(* IEC 61131-3 sources: volt/packages/volt-lsp-iec/test-corpus/lenze-mid/Device/Plc Logic/Application/Library Manager/L_OEEA_MachinePerformanceSolution, 3.26.4.18 (Lenze), 18 files *)

(* ---- SCCUTTHROUGPUTAVERAGELREAL.dut ---- *)
TYPE SCCUTTHROUGPUTAVERAGELREAL :
STRUCT
	LRREALINPUTVALUE : LREAL;
	LRINAVGVALUE : LREAL;
	SCUTREALSTR : STRING;
	LRCUTREAL : LREAL;
	IARRAYINDEX : INT;
	ALRVALUEARRAY : ARRAY [0..60] OF LREAL;
	LRAVERAGEVALUE : LREAL;
	LRLASTREALVALUE : LREAL;
	XARRAYFILLEDONCE : BOOL;
END_STRUCT
END_TYPE

(* ---- SCTREND_LIMITS.dut ---- *)
TYPE SCTREND_LIMITS :
STRUCT
	LRUPPERLIMIT : LREAL;
	DIUPPERROUNDLIMIT : DINT;
	DIMIDDLEROUNDLIMIT : DINT;
	DIFACTOR : INT;
	XTARGETUPPER : BOOL;
END_STRUCT
END_TYPE

(* ---- VERSIONCONSTANTS.gvl ---- *)
VAR_GLOBAL
	GC_BYAMOUNTOFGENERALDATA : BYTE := 50;
	GC_BYAMOUNTDOWNTIMEERRORS : BYTE := 10;
	GC_IFILTERSAMPLES : INT := 20;
END_VAR

(* ---- CALACTUALALLTIME.pou ---- *)
FUNCTION CALACTUALALLTIME : TIME
VAR_INPUT
	DTCURRENTTIME : TIME_OF_DAY;
	DTSETWEEKSTARTTIME : TIME_OF_DAY;
	EACTUALWEEKDAY : RTCLK.WEEKDAY;
	ESETWEEKDAY : RTCLK.WEEKDAY;
END_VAR
END_FUNCTION

(* ---- CALAVERARGELREALSUMMERYVALUE.pou ---- *)
FUNCTION CALAVERARGELREALSUMMERYVALUE : LREAL
VAR_INPUT
	LRVALUE : LREAL;
	INOOFAVERAGECOUNT : INT;
END_VAR
VAR_IN_OUT
	SCCUTAVERAGEREAL : scCutThrougputAveragelReal;
END_VAR
END_FUNCTION

(* ---- XYTRENDUPPERLIMIT.pou ---- *)
FUNCTION XYTRENDUPPERLIMIT : scTrend_Limits
VAR_INPUT
	LRTARGETVALUE : LREAL;
	LRACTUALVALUE : LREAL;
END_VAR
END_FUNCTION

(* ---- FBPROLONGTIME.pou ---- *)
FUNCTION_BLOCK FBPROLONGTIME
VAR_INPUT
	TPROLONGTIME : TIME;
	XSTARTPROLONGTIME : BOOL;
END_VAR
VAR_OUTPUT
	XPROLONG : BOOL;
END_VAR
VAR
	TONPROLONGTIMER : TON;
	TRIGPROLONG : R_TRIG;
END_VAR
END_FUNCTION_BLOCK

(* ---- L_OEEA_BASE.pou ---- *)
FUNCTION_BLOCK L_OEEA_BASE
VAR_INPUT
	XENABLE : BOOL;
	XRESET : BOOL;
END_VAR
VAR_IN_OUT
	SCSHIFTVALUES : scCurrentShiftValues;
	SCPDINTERNAL : scInternalVar;
END_VAR
VAR
	XACTIVELICENSE : BOOL := TRUE;
	XFIRSTCYCLE : BOOL := FALSE;
	I : INT;
	SCSHIFTCHANGEPERFORMANCE : scPerformance_base;
	SCSHIFTCHANGESCAP : scAccessPoints;
	SCINTERNSHIFTVALUES : scCurrentShiftValues;
	PUIHOUR : UINT;
	PUIHOUR2 : UINT;
	PUIHOUR3 : UINT;
	PUIHOUR4 : UINT;
	PUIHOUR5 : UINT;
	PUIMINUTE : UINT;
	PUIMINUTE2 : UINT;
	PUIMINUTE3 : UINT;
	PUIMINUTE4 : UINT;
	PUIMINUTE5 : UINT;
	PUISECOND : UINT;
	PUISECOND2 : UINT;
	PUISECOND3 : UINT;
	PUISECOND4 : UINT;
	PUISECOND5 : UINT;
	PUIMILLISECOND : UINT;
	PUIMILLISECOND2 : UINT;
	PUIMILLISECOND3 : UINT;
	PUIMILLISECOND4 : UINT;
	PUIMILLISECOND5 : UINT;
	XERROR : DTU.Error;
	XERROR2 : DTU.Error;
	XERROR3 : DTU.Error;
	LRPROGRESSIVETARGET : LREAL;
	SCPDINTERNALCLEAR : scInternalVar;
	XSHIFTRESET : BOOL;
	XINCONSISTENTDATARESET : BOOL;
	DTDAYCHANGETIME : TIME_OF_DAY;
	DTSTARTRECORDDATETIME : DATE_AND_TIME := DATE_AND_TIME#1970-1-1-0:0;
	FTXACTIVESHIFT : F_TRIG;
	FT_XRESET : R_TRIG;
	RTSHIFT0 : R_TRIG;
	RS_XRESET : RS;
	RTDOWNTIMECOUNT : R_TRIG;
	RTCALLFORSERVICE : R_TRIG;
	FBRRTIMER : TON;
	FBCALLFORSERVICE : TON;
	FBOEEKPISTIMEEVENT : TON;
	FBOEEKPIPROLONGED : TON;
	ILASTPRODUCTIONMODE : INT;
	ILASTDOWNTIMECATEGORY : INT;
	IPREVPRODUCTIONMODE : INT;
	IPREVDOWNTIMECATEGORY : INT;
	UDILASTDOWNTIMEREASON : UDINT;
	UDIPREVDOWNTIMEREASON : UDINT;
	IWEEKDAYDIFF : INT;
	XDEACTIVESHIFTCONTINIOUSUPDATE : BOOL;
	XSHIFTRESETEVENTDELAY : BOOL;
	XSHIFTRESETEVENTDELAYDONE : BOOL;
	FBACTUALPARTCOUNT : TON_Pausable;
	XRESETPRODUCTTYPEDATA : BOOL;
	T100MSTIMER : TON;
	DTCURRENTTIME : TIME_OF_DAY;
	XSTATECHANGEDETECTED : BOOL;
	FTRIGENDWAITINGTIMEPOWERONCYCLE : F_TRIG;
	RLASTTECHNICALCYCLETIME : REAL;
	RPARTTARGET_ACT : REAL;
	RTIMEDELTA : REAL;
	RLASTTARGETOEE : REAL;
	XSTATECHANGEAFTERPOWERCYCLE : BOOL;
	FBSTATECHANGEAFTERPOWERCYCLE : TON;
	XSTATECHANGEWAITINGTIME : BOOL;
	XSTATECHANGEDETECTEDONECYCLE : BOOL;
	SCIN_BATCHPRODUCTEND : scBatchProductEnd;
	SCBATCHPRODUCTEND : scBatchProductEnd;
	XFTXACTIVESHIFTDETECTED : BOOL;
	XHALTTIMETRIGGER : BOOL;
	THALTTIMETRIGGER : TIME;
	TONPROLONGTIMER : ARRAY [1..2] OF TON;
	ISTEPSHIFTCHANGE : INT := 0;
	XEVENTPROLONG : BOOL;
	XWAITPROLONG : BOOL;
	XSTATECHANGEPROLONGED : BOOL;
	FBSTATECHANGE : fbProlongTime;
	FBSTATECHANGEWAIT : fbProlongTime;
	XSEQSTATECHANGEBUSY : BOOL;
	XPRODUCTIONEVENTMODE : BOOL;
	XRESETDEACTIVESHIFTCONTINIOUSUPDATE : BOOL;
	XSETDEACTIVESHIFTCONTINIOUSUPDATE : BOOL;
END_VAR
END_FUNCTION_BLOCK

METHOD ACT_MAIN_BASE : BOOL
VAR_INPUT
	SCTRIGGER : scTrigger_base;
	EOEECALCMODE : enumOEECalculationMode;
	IPRODUCTIONEVENTMODE : INT;
END_VAR
VAR_IN_OUT
	SCMACHINEDATA : scMachineData_base;
	SCSHIFTVALUES : scCurrentShiftValues;
	SCSHIFTPERFORMANCE : scPerformance_base;
	SCPDINTERNAL : scInternalVar;
END_VAR
END_METHOD

METHOD ACT_PARTCOUNTER : BOOL
VAR_IN_OUT
	SCMACHINEDATA : scMachineData_base;
	SCSHIFTVALUES : scCurrentShiftValues;
	SCSHIFTPERFORMANCE : scPerformance_base;
	SCPDINTERNAL : scInternalVar;
END_VAR
END_METHOD

METHOD ACT_SHIFTCHANGEEVENT : BOOL
VAR_IN_OUT
	SCMACHINEDATA : scMachineData_base;
	SCSHIFTVALUES : scCurrentShiftValues;
	SCSHIFTPERFORMANCE : scPerformance_base;
	SCPDINTERNAL : scInternalVar;
END_VAR
END_METHOD

METHOD CAL_PRODUCTIONLOSSES : BOOL
VAR_INPUT
	EOEECALCMODE : enumOEECalculationMode;
END_VAR
VAR_IN_OUT
	SCMACHINEDATA : scMachineData_base;
	SCSHIFTVALUES : scCurrentShiftValues;
	SCPDINTERNAL : scInternalVar;
END_VAR
END_METHOD

METHOD SET_SHIFTDATA : BOOL
VAR_INPUT
	SCTRIGGER : scTrigger_base;
	IPRODUCTIONEVENTMODE : INT;
END_VAR
VAR_IN_OUT
	SCMACHINEDATA : scMachineData_base;
	SCSHIFTVALUES : scCurrentShiftValues;
	SCSHIFTPERFORMANCE : scPerformance_base;
	SCPDINTERNAL : scInternalVar;
END_VAR
END_METHOD

METHOD CAL_PRODUCTIONKPIS : BOOL
VAR_INPUT
	EOEECALCMODE : enumOEECalculationMode;
END_VAR
VAR_IN_OUT
	SCMACHINEDATA : scMachineData_base;
	SCSHIFTPERFORMANCE : scPerformance_base;
	SCPDINTERNAL : scInternalVar;
END_VAR
END_METHOD

METHOD METH_PROLONGBIT : BOOL
VAR_INPUT
	TPROLONGTIME : TIME;
END_VAR
VAR_IN_OUT
	TONPROLONGTIMER : TON;
	XSTARTPROLONGTIME : BOOL;
END_VAR
END_METHOD

(* ---- L_OEEA_CLOUDIF_NA.pou ---- *)
FUNCTION_BLOCK L_OEEA_CLOUDIF_NA
VAR_INPUT
	SDOWNTIMEBITSTR : STRING;
	SCTRIGGER : scTrigger;
	XENABLE : BOOL;
END_VAR
VAR_OUTPUT
	SCCLOUD : scCloud;
END_VAR
VAR_IN_OUT
	SCMACHINEDATA : scMachineData;
	SCPERFORMANCE : scPerformance;
END_VAR
VAR
	FBTRIGGER_SETTINGS : TON;
	FBTRIGGER_RR : TON;
	FBTRIGGER2_SETTINGS : TON;
	FBTRIGGER2_RR : TON;
	FBFIRSTSTARTTRIGGER : TON;
	XFIRSTCYCLE : BOOL;
	XFIRSTTRIGGER : BOOL;
END_VAR
END_FUNCTION_BLOCK

METHOD ACT_MAPVARIABLE
END_METHOD

METHOD ACT_TRIGGERVARIABLE
END_METHOD

(* ---- L_OEEA_DATASIMULATOR.pou ---- *)
FUNCTION_BLOCK L_OEEA_DATASIMULATOR
VAR_INPUT
	XENABLE : BOOL;
	PA_TIMER : RT_Timer;
	XMATERIALPRODUCTION : BOOL;
	RLINESPEED : REAL;
	IPARTCOUNTNOK : INT;
	IINPRODUCTIONMODE : INT;
	INOOFERRORINDEX : INT;
	LRMATERIALCOUNT : LREAL;
END_VAR
VAR_IN_OUT
	SCRT_STATUS_RECORD : RT_Status_Struct;
	SCSHIFTVALUES : scCurrentShiftValues;
	PA_DOWNTIME : RT_Downtime;
END_VAR
VAR
	FBTONALIVE : TON;
	FBR_TRIG_ALIVE : R_TRIG;
	FBTONOK_PARTS : TON;
	FBR_TRIG_OK_PARTS : R_TRIG;
	FBTONNOK_PARTS : TON;
	FBR_TRIG_NOK_PARTS : R_TRIG;
	FBTONERROR : TON;
	FBTONERRORDURATION : TON;
	FBTONPARTCYCLETIME : TON;
	FBTONOPCYCLETIME : TON;
	ERROR_INDEX : INT := 0;
	XERRORDETECTED : BOOL;
	LRAVERAGECYCLETIME : LREAL;
	DICOUNTCYCLETIMES : DINT;
	LRRANDOM : LREAL := 0.3287643289;
	IPARTCOUNTOK : INT;
	XTEST : BOOL;
	PREVXSCHEDULEDDOWNTIME : BOOL;
	TOK_PART : TIME;
	LRLASTMATERIALCOUNT : LREAL;
END_VAR
END_FUNCTION_BLOCK

METHOD CALC_PARTCOUNTER
END_METHOD

METHOD CALC_ALIVECOUNTER
END_METHOD

METHOD CALC_DOWNTIME
END_METHOD

METHOD CALC_MACHINECYCLETIME
END_METHOD

METHOD SET_PARTTYPE
END_METHOD

METHOD SET_PRODUCTIONMODE
END_METHOD

(* ---- L_OEEA_MACHINEPERFORMANCE.pou ---- *)
FUNCTION_BLOCK L_OEEA_MACHINEPERFORMANCE EXTENDS L_OEEA_Base
VAR_INPUT
	SCTRIGGER : scTrigger;
	XUPDATEJSONOEEKPI : BOOL;
	SPOWERUPJSONSUBSTR : STRING(255);
END_VAR
VAR_IN_OUT
	SCMACHINEDATA : scMachineData;
	SCSHIFTPERFORMANCE : scPerformance;
END_VAR
VAR
	FBTRIGGER_SETTINGS : TON;
	FBTRIGGER_RR : TON;
	FBTRIGGER2_SETTINGS : TON;
	FBTRIGGER2_RR : TON;
	FBCHANGEOVERTIMEEXCEEDED : TON;
	FBCHANGEOVERTIMEACTIVE : TP;
	IPREVIOUSSHIFT : INT;
	FBPRODUCTDATAPROLONGED : TON;
	FBLINESPEEDPROLONGED : TON;
	DILASTJOBID : DINT;
	RLASTACTUALSPEEDPERCENT : REAL;
	RLASTACTUALSPEEDVALUE : REAL;
	RPREVIOUSLASTCYCLETIME : REAL;
	RTMIDNIGHT : R_TRIG;
	SCTHROUGHPUTCLEAR : scThroughput;
	DILASTACTUALRUNTIME : DINT;
	DIACTUALUSEDTIME : DINT;
	SCAVERARGEHOURLYQUANTITY : scCutThrougputAverageLReal;
	SCAVERARGEHOURLYTARGET : scCutThrougputAverageLReal;
	SCSHIFTRESET : scCutThrougputAverageLReal;
	UI_1MINRUNTIME : UINT;
	LRLASTACTUALQUANTITYOK : LREAL;
	RLASTTARGETQUANTITYOK : REAL;
	RPREVIOUSTARGETOEE : REAL;
	RPREVIOUSTECHNICALCYCLETIME : REAL;
	ILENGHTOFJSONSTRING : INT;
	RTSTATCHANGEDETECT : R_TRIG;
	LRMAXACTUALTARGET : LREAL;
	LRMAXACTUALVALUE : LREAL;
	RTUPDATEJSONOEEKPI : R_TRIG;
	XACTUALARRAYFILLEDONCE : BOOL;
	XACTUALARRAYFILLEDONCEOUT : BOOL;
	XTARGETARRAYFILLEDONCE : BOOL;
	XTARGETARRAYFILLEDONCEOUT : BOOL;
	IAVERAGEARRAYLENGHT : INT := 60;
	ICALCTHROUGHPUT : INT := 0;
	IFIRSTMODEEVENT : INT;
	ISHIFTEVENT : INT;
	ISHIFTPRODUCTEVENT : INT;
	RTSHIFTDAYSTARTPROLONG : R_TRIG;
	RTSHIFTDAYENDPROLONG : R_TRIG;
	XRESETBATCHIDDATA : BOOL;
	XWAITFORPOWERUPCYCLEEND : BOOL;
	FBUPDATEJSONOEEKPIINPUT : TON;
	XUPDATEJSONOEEKPIDETECTED : BOOL;
	XTRIGGER_SETTINGS_PLCCYCLDELAY : BOOL;
	XFTXACTIVESHIFTDETECTED2 : BOOL;
	ISETCALCTHROUGHPUT : INT;
END_VAR
END_FUNCTION_BLOCK

METHOD CAL_RUNRATE
END_METHOD

METHOD ACT_BUTTONS
END_METHOD

METHOD ACT_PRODUCTIONKPIS_EXTENDED
END_METHOD

METHOD ACT_SHIFTDATA_EXTENDED
END_METHOD

METHOD ACT_SHIFTCHANGEEVENT_EXTENDED
END_METHOD

METHOD ACT_CREATEJSONPRODUCTOEEKPIDATA
END_METHOD

METHOD ACT_CREATEJSONEVENTDATA
END_METHOD

(* ---- L_OEEA_MACHINEPERFORMANCE_BASE.pou ---- *)
FUNCTION_BLOCK L_OEEA_MACHINEPERFORMANCE_BASE EXTENDS L_OEEA_Base
VAR_INPUT
	SCTRIGGER : scTrigger_base;
END_VAR
VAR_IN_OUT
	SCMACHINEDATA : scMachineData_base;
	SCSHIFTPERFORMANCE : scPerformance_base;
END_VAR
END_FUNCTION_BLOCK

(* ---- L_OEEA_PERFORMANCEDASHBOARD_NA.pou ---- *)
FUNCTION_BLOCK L_OEEA_PERFORMANCEDASHBOARD_NA
VAR_INPUT
	XENABLE : BOOL;
	XRESETHISTORY : BOOL;
END_VAR
VAR_IN_OUT
	SCSHIFTVALUES : scCurrentShiftValues;
	SCSHIFTPERFORMANCE : scPerformance;
	SCDOWNTIME : scDowntime;
	SCPDSHIFTHISTORY : scVisuShiftHistory;
	SCPERFORMANCEDASHBOARD : scVisuPerformanceDashboard;
END_VAR
VAR
	I : INT;
	SCRESETSHIFTHISTORY : scVisuShiftHistory;
END_VAR
END_FUNCTION_BLOCK

METHOD ACT_MAPVARIABLE
END_METHOD

METHOD ACT_PRODUCTIONSTATUS
END_METHOD

(* ---- L_OEEA_SHIFTOEEHISTORY.pou ---- *)
FUNCTION_BLOCK L_OEEA_SHIFTOEEHISTORY
VAR_INPUT
	XENABLE : BOOL;
	XRESETHISTORY : BOOL;
END_VAR
VAR_IN_OUT
	SCSHIFTPERFORMANCE : scPerformance;
	SCSHIFTVALUES : scCurrentShiftValues;
	SCSHIFTHISTORY : ARRAY [1..3] OF scPerformance;
END_VAR
VAR
	SCSHIFTCHANGEPERFORMANCE : scPerformance;
	I : INT;
	ISHFTCHANGECOUNTER : INT;
END_VAR
END_FUNCTION_BLOCK

(* ---- L_OEEA_SHIFTOEEHISTORY_BASE.pou ---- *)
FUNCTION_BLOCK L_OEEA_SHIFTOEEHISTORY_BASE
VAR_INPUT
	XENABLE : BOOL;
	XRESETHISTORY : BOOL;
END_VAR
VAR_IN_OUT
	SCSHIFTVALUES : scCurrentShiftValues;
	SCSHIFTPERFORMANCE : scPerformance_base;
	SCPDSHIFTHISTORY : scVisuShiftHistory_base;
END_VAR
VAR
	I : INT;
	SCRESETSHIFTHISTORY : scVisuShiftHistory_base;
	XFIRSTPOWERUPCYCLEENDS : BOOL;
	XFIRSTPLCCYCLE : BOOL;
	FTRIG_POWERONCYCLEPROLONGED : F_TRIG;
END_VAR
END_FUNCTION_BLOCK

(* ---- L_OEEA_X_TREND.pou ---- *)
FUNCTION_BLOCK L_OEEA_X_TREND
VAR_INPUT
	XENABLE : BOOL;
	XTRIGGER : BOOL;
	XSORTUPDOWN : BOOL;
	X_AXIS_VALUE : DATE_AND_TIME;
END_VAR
VAR_OUTPUT
	XTRIGGERSYNC : BOOL;
END_VAR
VAR_IN_OUT
	X_AXIS_TREND : ARRAY [0..GVL_Const_Production_log.imaxSizeXY_TREND] OF DATE_AND_TIME;
	X2_AXIS_TREND : ARRAY [0..GVL_Const_Production_log.imaxSizeXY_TREND] OF DINT;
	X3_AXIS_TREND : ARRAY [0..GVL_Const_Production_log.imaxSizeXY_TREND] OF INT;
END_VAR
VAR
	I : INT;
	IMAXSIZE : INT;
	XRESET_Y_TREND_TRIG : R_TRIG;
	DIX2VALUE : DINT;
	R_TRIG_TRIGGERSYNC : R_TRIG;
	XFIRST_CYCLE : BOOL;
END_VAR
END_FUNCTION_BLOCK

(* ---- L_OEEA_Y_TREND.pou ---- *)
FUNCTION_BLOCK L_OEEA_Y_TREND
VAR_INPUT
	XENABLE : BOOL;
	XTRIGGER : BOOL;
	XSORTUPDOWN : BOOL;
	Y_AXIS_ACTUAL_VALUE : LREAL;
	Y_AXIS_TARGET_VALUE : LREAL;
	XRESET_Y_TREND : BOOL;
END_VAR
VAR_OUTPUT
	XVALUECHANGE : BOOL;
	SCTREND_LIMITS : scTrend_Limits;
END_VAR
VAR_IN_OUT
	Y_AXIS_TREND : ARRAY [0..GVL_Const_Production_log.imaxSizeXY_TREND] OF LREAL;
	Y_AXIS_TARGET : ARRAY [0..GVL_Const_Production_log.imaxSizeXY_TREND] OF LREAL;
END_VAR
VAR
	I : INT;
	IMAXSIZE : INT;
	XRESET_Y_TREND_TRIG : R_TRIG;
	Y_AXIS_VALUE_PREVIOUS : LREAL;
	LRAXISTARGETMAXVALUE : LREAL;
	LRAXISACTUALMAXVALUE : LREAL;
END_VAR
END_FUNCTION_BLOCK

(* ---- TON_PAUSABLE.pou ---- *)
FUNCTION_BLOCK TON_PAUSABLE
VAR_INPUT
	IN : BOOL;
	PT : TIME;
	PAUSE : BOOL;
END_VAR
VAR_OUTPUT
	Q : BOOL;
	ET : TIME;
END_VAR
VAR
	RTPAUSE : R_TRIG;
	TTIMEPAUSED : TIME;
	TON : TON;
END_VAR
END_FUNCTION_BLOCK
